(* IEC 61131-3 sources: RL_MAR/experiments/comparison/llm4plc/results/gpt-4o_20260507_114630/20260507_120353, 3 files *)

(* ---- generated_code_iteration_0.st ---- *)
plaintext
START_ST
FUNCTION_BLOCK PrecisionEngravingMachine
VAR_INPUT
    DesignSelection : INT; // Input for the selected design
    EngravingDepth : REAL; // Input for engraving depth
    EngravingSpeed : REAL; // Input for engraving speed
END_VAR

VAR_OUTPUT
    ZAxisMotor : BOOL; // Output to control the Z-axis motor
    EngravingMotor : BOOL; // Output to control the engraving motor
END_VAR

VAR
    state : INT; // Current state of the system
    prevState : INT; // Previous state of the system to detect state changes
    CalculatedDepth : REAL; // Internal variable to store the calculated engraving depth
    CalculatedSpeed : REAL; // Internal variable to store the calculated engraving speed
END_VAR

// State Definitions
// STATE 0: IDLE
// STATE 1: CONFIGURE DESIGN PARAMETERS
// STATE 2: ACTIVATE MOTORS
// STATE 3: INVALID DESIGN

// Initialization
IF (state = 0) AND (prevState = 0) THEN
    // Set initial state to IDLE
    state := 0;
    prevState := 0;
    ZAxisMotor := FALSE;
    EngravingMotor := FALSE;
    CalculatedDepth := 0.0;
    CalculatedSpeed := 0.0;
ENDIF;

// State Machine Logic
CASE state OF
    // STATE 0: IDLE
    0:
        ZAxisMotor := FALSE;
        EngravingMotor := FALSE;
        CalculatedDepth := 0.0;
        CalculatedSpeed := 0.0;

        // Transition to STATE 1 if a valid design is selected
        IF DesignSelection IN [1, 2, 3] THEN
            state := 1;
        END_IF;

    // STATE 1: CONFIGURE DESIGN PARAMETERS
    1:
        ZAxisMotor := FALSE;
        EngravingMotor := FALSE;

        // Configure engraving parameters based on design selection
        CASE DesignSelection OF
            1:
                CalculatedDepth := 0.1;
                CalculatedSpeed := 10.0;
            2:
                CalculatedDepth := 0.2;
                CalculatedSpeed := 8.0;
            3:
                CalculatedDepth := 0.15;
                CalculatedSpeed := 12.0;
        ELSE
            // Transition to STATE 3 if invalid design is selected
            state := 3;
        END_CASE;

        // Transition to STATE 2 if a valid design is selected
        IF DesignSelection IN [1, 2, 3] THEN
            state := 2;
        END_IF;

    // STATE 2: ACTIVATE MOTORS
    2:
        ZAxisMotor := TRUE;
        EngravingMotor := TRUE;

        // Retain the calculated depth and speed
        EngravingDepth := CalculatedDepth;
        EngravingSpeed := CalculatedSpeed;

        // Transition to STATE 1 if design changes to another valid design
        IF (DesignSelection IN [1, 2, 3]) AND (DesignSelection <> prevState) THEN
            state := 1;
        END_IF;

        // Transition to STATE 3 if design changes to an invalid design
        IF DesignSelection NOT IN [1, 2, 3] THEN
            state := 3;
        END_IF;

    // STATE 3: INVALID DESIGN
    3:
        ZAxisMotor := FALSE;
        EngravingMotor := FALSE;
        CalculatedDepth := 0.0;
        CalculatedSpeed := 0.0;

        // Transition to STATE 1 if a valid design is selected
        IF DesignSelection IN [1, 2, 3] THEN
            state := 1;
        END_IF;
END_CASE;

// Update previous state
prevState := state;

END_FUNCTION_BLOCK
END_ST

(* ---- generated_code_iteration_1.st ---- *)
START_REASON
The feedback indicates that the issue lies in the improper use of `IF` statements, specifically the lack of proper termination with `ELSIF`, `ELSE`, or `END_IF`. This likely occurs in one or more places where `IF` statements are used without a corresponding `END_IF` or proper structure. This could lead to a failure in the CODESYS compiler validation.

To address this, I will carefully review all `IF` statements in the code and ensure they are properly terminated and structured. Additionally, I will verify the overall logic to ensure correctness and compliance with syntax rules.
END_REASON

START_ST
FUNCTION_BLOCK PrecisionEngravingMachine
VAR_INPUT
    DesignSelection : INT; // Input for the selected design
    EngravingDepth : REAL; // Input for engraving depth
    EngravingSpeed : REAL; // Input for engraving speed
END_VAR

VAR_OUTPUT
    ZAxisMotor : BOOL; // Output to control the Z-axis motor
    EngravingMotor : BOOL; // Output to control the engraving motor
END_VAR

VAR
    state : INT; // Current state of the system
    prevState : INT; // Previous state of the system to detect state changes
    CalculatedDepth : REAL; // Internal variable to store the calculated engraving depth
    CalculatedSpeed : REAL; // Internal variable to store the calculated engraving speed
END_VAR

// State Definitions
// STATE 0: IDLE
// STATE 1: CONFIGURE DESIGN PARAMETERS
// STATE 2: ACTIVATE MOTORS
// STATE 3: INVALID DESIGN

// Initialization
IF (state = 0) AND (prevState = 0) THEN
    // Set initial state to IDLE
    state := 0;
    prevState := 0;
    ZAxisMotor := FALSE;
    EngravingMotor := FALSE;
    CalculatedDepth := 0.0;
    CalculatedSpeed := 0.0;
END_IF;

// State Machine Logic
CASE state OF
    // STATE 0: IDLE
    0:
        ZAxisMotor := FALSE;
        EngravingMotor := FALSE;
        CalculatedDepth := 0.0;
        CalculatedSpeed := 0.0;

        // Transition to STATE 1 if a valid design is selected
        IF DesignSelection IN [1, 2, 3] THEN
            state := 1;
        END_IF;

    // STATE 1: CONFIGURE DESIGN PARAMETERS
    1:
        ZAxisMotor := FALSE;
        EngravingMotor := FALSE;

        // Configure engraving parameters based on design selection
        CASE DesignSelection OF
            1:
                CalculatedDepth := 0.1;
                CalculatedSpeed := 10.0;
            2:
                CalculatedDepth := 0.2;
                CalculatedSpeed := 8.0;
            3:
                CalculatedDepth := 0.15;
                CalculatedSpeed := 12.0;
            ELSE
                // Transition to STATE 3 if invalid design is selected
                state := 3;
        END_CASE;

        // Transition to STATE 2 if a valid design is selected
        IF DesignSelection IN [1, 2, 3] THEN
            state := 2;
        END_IF;

    // STATE 2: ACTIVATE MOTORS
    2:
        ZAxisMotor := TRUE;
        EngravingMotor := TRUE;

        // Retain the calculated depth and speed
        EngravingDepth := CalculatedDepth;
        EngravingSpeed := CalculatedSpeed;

        // Transition to STATE 1 if design changes to another valid design
        IF (DesignSelection IN [1, 2, 3]) AND (DesignSelection <> prevState) THEN
            state := 1;
        ELSIF DesignSelection NOT IN [1, 2, 3] THEN
            // Transition to STATE 3 if design changes to an invalid design
            state := 3;
        END_IF;

    // STATE 3: INVALID DESIGN
    3:
        ZAxisMotor := FALSE;
        EngravingMotor := FALSE;
        CalculatedDepth := 0.0;
        CalculatedSpeed := 0.0;

        // Transition to STATE 1 if a valid design is selected
        IF DesignSelection IN [1, 2, 3] THEN
            state := 1;
        END_IF;
END_CASE;

// Update previous state
prevState := state;

END_FUNCTION_BLOCK
END_ST

(* ---- generated_code_iteration_2.st ---- *)
START_REASON
The feedback indicates that the issue lies in the improper use of the `IN` keyword in `IF` statements. Specifically, the `IN` keyword is not valid in CODESYS Structured Text syntax for checking membership in a set or range. Instead, the correct approach is to use logical operators such as `AND` and `OR` to construct equivalent conditions.

To address this, I will replace all instances of `IN` with appropriate logical conditions using `AND` and `OR`. Additionally, I will verify the overall logic to ensure correctness and compliance with CODESYS syntax rules.
END_REASON

START_ST
FUNCTION_BLOCK PrecisionEngravingMachine
VAR_INPUT
    DesignSelection : INT; // Input for the selected design
    EngravingDepth : REAL; // Input for engraving depth
    EngravingSpeed : REAL; // Input for engraving speed
END_VAR

VAR_OUTPUT
    ZAxisMotor : BOOL; // Output to control the Z-axis motor
    EngravingMotor : BOOL; // Output to control the engraving motor
END_VAR

VAR
    state : INT; // Current state of the system
    prevState : INT; // Previous state of the system to detect state changes
    CalculatedDepth : REAL; // Internal variable to store the calculated engraving depth
    CalculatedSpeed : REAL; // Internal variable to store the calculated engraving speed
END_VAR

// State Definitions
// STATE 0: IDLE
// STATE 1: CONFIGURE DESIGN PARAMETERS
// STATE 2: ACTIVATE MOTORS
// STATE 3: INVALID DESIGN

// Initialization
IF (state = 0) AND (prevState = 0) THEN
    // Set initial state to IDLE
    state := 0;
    prevState := 0;
    ZAxisMotor := FALSE;
    EngravingMotor := FALSE;
    CalculatedDepth := 0.0;
    CalculatedSpeed := 0.0;
END_IF;

// State Machine Logic
CASE state OF
    // STATE 0: IDLE
    0:
        ZAxisMotor := FALSE;
        EngravingMotor := FALSE;
        CalculatedDepth := 0.0;
        CalculatedSpeed := 0.0;

        // Transition to STATE 1 if a valid design is selected
        IF (DesignSelection = 1) OR (DesignSelection = 2) OR (DesignSelection = 3) THEN
            state := 1;
        END_IF;

    // STATE 1: CONFIGURE DESIGN PARAMETERS
    1:
        ZAxisMotor := FALSE;
        EngravingMotor := FALSE;

        // Configure engraving parameters based on design selection
        CASE DesignSelection OF
            1:
                CalculatedDepth := 0.1;
                CalculatedSpeed := 10.0;
            2:
                CalculatedDepth := 0.2;
                CalculatedSpeed := 8.0;
            3:
                CalculatedDepth := 0.15;
                CalculatedSpeed := 12.0;
            ELSE
                // Transition to STATE 3 if invalid design is selected
                state := 3;
        END_CASE;

        // Transition to STATE 2 if a valid design is selected
        IF (DesignSelection = 1) OR (DesignSelection = 2) OR (DesignSelection = 3) THEN
            state := 2;
        END_IF;

    // STATE 2: ACTIVATE MOTORS
    2:
        ZAxisMotor := TRUE;
        EngravingMotor := TRUE;

        // Retain the calculated depth and speed
        EngravingDepth := CalculatedDepth;
        EngravingSpeed := CalculatedSpeed;

        // Transition to STATE 1 if design changes to another valid design
        IF ((DesignSelection = 1) OR (DesignSelection = 2) OR (DesignSelection = 3)) AND (DesignSelection <> prevState) THEN
            state := 1;
        ELSIF NOT ((DesignSelection = 1) OR (DesignSelection = 2) OR (DesignSelection = 3)) THEN
            // Transition to STATE 3 if design changes to an invalid design
            state := 3;
        END_IF;

    // STATE 3: INVALID DESIGN
    3:
        ZAxisMotor := FALSE;
        EngravingMotor := FALSE;
        CalculatedDepth := 0.0;
        CalculatedSpeed := 0.0;

        // Transition to STATE 1 if a valid design is selected
        IF (DesignSelection = 1) OR (DesignSelection = 2) OR (DesignSelection = 3) THEN
            state := 1;
        END_IF;
END_CASE;

// Update previous state
prevState := state;

END_FUNCTION_BLOCK
END_ST
